(* PLC project CodesysTest_empty.project, CODESYS CODESYS V3.5 SP17 Patch 3 *)
(* stored: creationDateTime 2022-04-23T16:32:03.491546, modificationDateTime 2022-04-22T11:58:57.9681441 *)

CONFIGURATION Application
  RESOURCE Application ON PLC
    TASK MainTask(INTERVAL := T#200ms, PRIORITY := 1);
  END_RESOURCE
END_CONFIGURATION
